# EPICS autosave request: iocBoot/ioc13ida_E_Mono_XPS/auto_positions.req
file "CARS_motor_positions.req",         P=$(P), M=m61
file "CARS_motor_positions.req",         P=$(P), M=m62
file "CARS_motor_positions.req",         P=$(P), M=m63
file "CARS_motor_positions.req",         P=$(P), M=m64
file "CARS_motor_positions.req",         P=$(P), M=m65
file "CARS_motor_positions.req",         P=$(P), M=m66
file "CARS_motor_positions.req",         P=$(P), M=m67
file "CARS_motor_positions.req",         P=$(P), M=m68
